# EPICS StreamDevice protocol: protocols/slowmon.proto
# slowmon controls.
Terminator = LF;
ExtraInput = Ignore;

setNACC {
	out "nacc %(A)d,%(B)d,%(C)d,%(D)d";
	in;
}

setDNA {
	out "dna %d";
	in;
}

getDNA {
	out "dna";
	in "%d";
}

setSlowmonFs {
	out "slowmon_fs %d";
	in;
}

setSlowmonFin {
	out "slowmon_fin %d";
	in;
}
